FUNCTION_BLOCK PUBLIC PAETurnHeadDist EXTENDS PAEEMotor2D
VAR_INPUT
END_VAR
VAR_OUTPUT
END_VAR
VAR
	_PAPointMatIn1 : PAPoint(THIS^);
	_PAPointMatOut01 : PAPoint(THIS^);
	_PAPointMatOut02 : PAPoint(THIS^);
	_PAPointMatOut03 : PAPoint(THIS^);
	_PAPointMatOut04 : PAPoint(THIS^);
	_PAPointMatOut05 : PAPoint(THIS^);
	_PAPointMatOut06 : PAPoint(THIS^);
	_PAPointMatOut07 : PAPoint(THIS^);
	_PAPointMatOut08 : PAPoint(THIS^);
	_PAPointMatOut09 : PAPoint(THIS^);
	_PAPointMatOut10 : PAPoint(THIS^);
	_DesiredPosition : INT;
	_Position : INT;
	_ReqPosition : INT;
END_VAR

{attribute 'monitoring' := 'call'}
//{attribute 'TcRpcEnable'}
PROPERTY PUBLIC DesiredPosition : INT
GET // PUBLIC
DesiredPosition := _DesiredPosition;
END_GET
SET // PUBLIC
_DesiredPosition := DesiredPosition;
Root.OnPropertyChangedInt(THIS^, 56, _DesiredPosition);
END_SET
END_PROPERTY

METHOD FB_init : BOOL
VAR_INPUT
	bInitRetains : BOOL; // if TRUE, the retain variables are initialized (warm start / cold start)
	bInCopyCode : BOOL;  // if TRUE, the instance afterwards gets moved into the copy code (online change)
	parent : IACComponent;
END_VAR
AddPoint(_PAPointMatIn1);
AddPoint(_PAPointMatOut01);
AddPoint(_PAPointMatOut02);
AddPoint(_PAPointMatOut03);
AddPoint(_PAPointMatOut04);
AddPoint(_PAPointMatOut05);
AddPoint(_PAPointMatOut06);
AddPoint(_PAPointMatOut07);
AddPoint(_PAPointMatOut08);
AddPoint(_PAPointMatOut09);
AddPoint(_PAPointMatOut10);
END_METHOD

METHOD FB_postinit
VAR_INPUT
	root : IACVariobatch;
END_VAR
SUPER^.FB_postinit(root);  
root.OnPropertyChangedInt(THIS^, 55, _Position);
root.OnPropertyChangedInt(THIS^, 56, _DesiredPosition);
root.OnPropertyChangedInt(THIS^, 57, _ReqPosition);
END_METHOD

METHOD PUBLIC HasPointReachedOffPosition : BOOL
VAR_INPUT
	point : IACPoint;
END_VAR
END_METHOD

METHOD PUBLIC HasPointReachedOnPosition : BOOL
VAR_INPUT
	point : IACPoint;
END_VAR
END_METHOD

METHOD PUBLIC InvokeSetterInt
VAR_INPUT
	PropertyID : INT;
	PropertyValue : INT;
END_VAR
SUPER^.InvokeSetterInt(PropertyID, PropertyValue);
CASE PropertyID OF
	55:
		Position := PropertyValue;
	56:
		DesiredPosition := PropertyValue;
	57:
		ReqPosition := PropertyValue;
END_CASE
END_METHOD

METHOD OnInitMemory
VAR_INPUT
	root : IACVariobatch;
END_VAR
RegisterProperty(root, 55, GCL.cSizeINT); //Position
RegisterProperty(root, 56, GCL.cSizeINT); //DesiredPosition
RegisterProperty(root, 57, GCL.cSizeINT); //ReqPosition
SUPER^.OnInitMemory(root);
END_METHOD

PROPERTY PUBLIC PAPointMatIn1 : IACPoint
GET // PUBLIC
PAPointMatIn1 := _PAPointMatIn1;
END_GET
END_PROPERTY

PROPERTY PUBLIC PAPointMatOut01 : IACPoint
GET // PUBLIC
PAPointMatOut01 := _PAPointMatOut01;
END_GET
END_PROPERTY

PROPERTY PUBLIC PAPointMatOut02 : IACPoint
GET // PUBLIC
PAPointMatOut02 := _PAPointMatOut02;
END_GET
END_PROPERTY

PROPERTY PUBLIC PAPointMatOut03 : IACPoint
GET // PUBLIC
PAPointMatOut03 := _PAPointMatOut03;
END_GET
END_PROPERTY

PROPERTY PUBLIC PAPointMatOut04 : IACPoint
GET // PUBLIC
PAPointMatOut04 := _PAPointMatOut04;
END_GET
END_PROPERTY

PROPERTY PUBLIC PAPointMatOut05 : IACPoint
GET
PAPointMatOut05 := _PAPointMatOut05;
END_GET
END_PROPERTY

PROPERTY PUBLIC PAPointMatOut06 : IACPoint
GET // PUBLIC
PAPointMatOut06 := _PAPointMatOut06;
END_GET
END_PROPERTY

PROPERTY PUBLIC PAPointMatOut07 : IACPoint
GET // PUBLIC
PAPointMatOut07 := _PAPointMatOut08;
END_GET
END_PROPERTY

PROPERTY PUBLIC PAPointMatOut08 : IACPoint
GET // PUBLIC
PAPointMatOut08 := _PAPointMatOut08;
END_GET
END_PROPERTY

PROPERTY PUBLIC PAPointMatOut09 : IACPoint
GET // PUBLIC
PAPointMatOut09 := _PAPointMatOut09;
END_GET
END_PROPERTY

PROPERTY PUBLIC PAPointMatOut10 : IACPoint
GET // PUBLIC
PAPointMatOut10 := _PAPointMatOut10;
END_GET
END_PROPERTY

{attribute 'monitoring' := 'call'}
//{attribute 'TcRpcEnable'}
PROPERTY PUBLIC Position : INT
GET // PUBLIC
Position := _Position;
END_GET
SET // PUBLIC
_Position := Position;
Root.OnPropertyChangedInt(THIS^, 55, _Position);
END_SET
END_PROPERTY

{attribute 'monitoring' := 'call'}
//{attribute 'TcRpcEnable'}
PROPERTY PUBLIC ReqPosition : INT
GET // PUBLIC
ReqPosition := _ReqPosition;
END_GET
SET // PUBLIC
_ReqPosition := ReqPosition;
Root.OnPropertyChangedInt(THIS^, 57, _ReqPosition);
IF Root.InSimulation THEN
	Position := _ReqPosition;
END_IF
END_SET
END_PROPERTY

METHOD PUBLIC TurnOnLeftWithPos
VAR_INPUT
END_VAR
END_METHOD

METHOD PUBLIC TurnOnRightWithPos
VAR_INPUT
END_VAR
END_METHOD

END_FUNCTION_BLOCK

(* stored: Version 1.1.0.1, ProductVersion 3.1.4024.6
   POU PAETurnHeadDist: Id {1791f932-5bf8-45fc-b4d6-be60ea6f55d1}, SpecialFunc None
   Property DesiredPosition: Id {4b5aa20c-ee37-4c63-8ff2-4dd5101ac2ba}
   Get Get: Id {704af908-372b-43e2-9257-ba39ce11f42c}
   Set Set: Id {36fd2fe3-0dbf-46b1-91d8-b69d81787cc0}
   Method FB_init: Id {00b03402-d621-4ff3-84a4-bc6d3c003a4f}
   Method FB_postinit: Id {b2a4cff4-e33d-4583-87a5-813c04828cb4}
   Method HasPointReachedOffPosition: Id {0b7dad62-5f36-4004-a118-40ae5df985f0}
   Method HasPointReachedOnPosition: Id {f6245a46-c667-4501-8412-ab0a826ec392}
   Method InvokeSetterInt: Id {76b3d27f-1106-43bb-ae3b-9cc3afc3307b}
   Method OnInitMemory: Id {c3468934-a1d9-4dbd-9411-f05d48e11033}
   Property PAPointMatIn1: Id {a404647b-5209-4499-9b58-b12891c06fa3}
   Get Get: Id {c0e8aedf-9ced-4017-b458-2a6cf7f9e560}
   Property PAPointMatOut01: Id {9a3cd5f6-e9d7-4e0e-9b27-ac3afd0b2f62}
   Get Get: Id {eb9be030-42cb-4474-bfab-34e559ce0f75}
   Property PAPointMatOut02: Id {2eb12494-70f4-4326-9c8a-b21b32bd3d99}
   Get Get: Id {f552503b-9579-4277-a2d8-99ce2e2275cc}
   Property PAPointMatOut03: Id {dcd48c1b-509d-42fa-ae95-2a57af204f4b}
   Get Get: Id {8690ca26-a8b3-4657-9456-b6f09f58417e}
   Property PAPointMatOut04: Id {3f4ce6c2-b659-422f-8665-cc674d6ec597}
   Get Get: Id {87516809-2aab-41fc-90fd-783c88a343df}
   Property PAPointMatOut05: Id {c2405e17-99f1-4c24-b38a-d635847f773f}
   Get Get: Id {0adab9bd-12e8-424a-9eaf-7dd9446c0e76}
   Property PAPointMatOut06: Id {8707f0d9-6a6b-47aa-bfff-a8480a21600a}
   Get Get: Id {3c6e12f1-e6fe-47c3-a081-5abcb8bb1030}
   Property PAPointMatOut07: Id {66f46587-d8d5-4445-bae7-99d5413d812a}
   Get Get: Id {c715ff0d-a285-4cb7-9004-39006b056fa9}
   Property PAPointMatOut08: Id {3eea5dee-07e5-481e-91e7-3e6f347a9a99}
   Get Get: Id {6eab18f3-3986-428d-a9ae-fee6dad82fa0}
   Property PAPointMatOut09: Id {4191852c-2db4-4cee-ae6a-f7c8e4a1ba38}
   Get Get: Id {0473c79f-9092-4b6d-9f63-6a142f884e66}
   Property PAPointMatOut10: Id {365fc2aa-81fc-4b42-92ee-2f247b889341}
   Get Get: Id {1c5240ec-75ce-4f82-ad2c-c6539a4416c4}
   Property Position: Id {3857d02a-e2dd-4115-82c9-7ced76ffdfa7}
   Get Get: Id {02533626-0fde-40d0-8742-2ea413334509}
   Set Set: Id {f295c1da-1e93-470b-a196-2458b496d9de}
   Property ReqPosition: Id {4bab6ba9-45b0-437f-ae11-62e7593c6fea}
   Get Get: Id {bcd011e1-e468-440b-b37d-ec6854eefe8c}
   Set Set: Id {e1441a23-e090-4f1a-86a2-13f15d0001a1}
   Method TurnOnLeftWithPos: Id {d2fc1164-7be0-4e86-b57f-4e1a9d584566}
   Method TurnOnRightWithPos: Id {9b4ce0de-df5d-4cef-80bd-2c040f7aaba6} *)
